(* CODESYS project distributedcontrol_1000.library
   Title: DistributedControl
   Version: 1.0.0.0
   Placeholder: DistributedControl
   Company: FactoryAutomation

Project tree, tasks and I/O mapping:
  libraries: Tc2_Standard, * (Beckhoff Automation GmbH); Tc2_System, * (Beckhoff Automation GmbH); Tc2_TcpIp, * (Beckhoff Automation GmbH); Tc3_Module, * (Beckhoff Automation GmbH)
  DUTs/
    data type E_TcpIpMode
    data type ST_ClientData
    data type ST_ServerData
  GVLs/
  POUs/
    program MAIN [ST]
    function block Payload [ST]
    function block Serializable [ST]: Deserialize, FB_exit, FB_init, Serialize
    function block TcpIp [ST]: FB_init, ReceiveSerializedObject, SendSerializedObject
  VISUs/
*)

// DUTs/E_TcpIpMode
TYPE E_TcpIpMode :
(
	TCP_IP_NO_MODE := 0,
	TCP_IP_SERVER,
	TCP_IP_CLIENT
);
END_TYPE

// DUTs/ST_ClientData
TYPE ST_ClientData :
STRUCT
	sSrvNetID   : T_AmsNetID := '';
    nMode       : DWORD := 0;
    sRemoteHost : T_IPv4Addr := '';
    nRemotePort : UDINT;
    tReconnect  : TIME := T#45S;
END_STRUCT
END_TYPE

// DUTs/ST_ServerData
TYPE ST_ServerData :
STRUCT
	hServer         : T_HSERVER; 
    sSrvNetID       : T_AmsNetID := ''; 
    sLocalHost      : STRING(15) := ''; 
    nLocalPort      : UDINT := 0;
	
    nMode           : DWORD := LISTEN_MODE_CLOSEALL (* OR CONNECT_MODE_ENABLEDBG*);
END_STRUCT
END_TYPE

// POUs/MAIN
PROGRAM MAIN
VAR

	fbPayload_1 : Payload(uiObjectSize := SIZEOF(Payload));
	fbPayload_2 : Payload(uiObjectSize := SIZEOF(Payload));
	
	bStart,
	bStart2,
	bStart3,
	bStart4,
	bStart5,
	bStart6 : BOOL;
	
	Size1,
	Size2,
	Size3,
	Size4 : UINT;
	pBuffer : POINTER TO BYTE;
	pServerBuffer : POINTER TO BYTE;
	pClientBuffer : POINTER TO BYTE;
	aMarshalBuffer : ARRAY[0..1999] OF BYTE;
	aServerMarshalBuffer : ARRAY[0..1999] OF BYTE;
	aClientMarshalBuffer : ARRAY[0..1999] OF BYTE;
	aServerBuffer : ARRAY[0..1999] OF BYTE;
	aClientBuffer : ARRAY[0..1999] OF BYTE;
	fbServer : TcpIp(TCP_IP_SERVER);
	fbClient : TcpIp(TCP_IP_CLIENT);
	serverStep : UINT;
	clientStep : UINT;
	udiServerTimeToSend : UDINT;
	udiServerTimeToReceive : UDINT;
	udiServerTimeToSendTmp : UDINT;
	udiServerTimeToReceiveTmp : UDINT;
END_VAR


fbPayload_1();
fbPayload_2();
fbPayload_1.timer.PT := T#45S;
fbPayload_1.timer.IN := TRUE;

fbServer.stServerData.nLocalPort := 200;
fbServer(bEnable := TRUE);

fbClient.stClientData.nRemotePort := 200;
fbClient(bEnable := TRUE);

IF 	bStart
	THEN
		
	pBuffer := fbPayload_2.Deserialize(fbPayload_1.Serialize());
	bStart := FALSE;
	
END_IF

IF	bStart2
	THEN
	
	MEMCPY(ADR(aMarshalBuffer),fbPayload_1.Serialize(),fbPayload_1.uiObjectSize);
	bStart2 := FALSE;
	
END_IF

IF	bStart3
	THEN
	
	fbPayload_2.Deserialize(ADR(aMarshalBuffer));
	bStart3 := FALSE;
	
END_IF

IF	bStart4
	THEN
	
	MEMCPY(ADR(aMarshalBuffer),fbPayload_2.Serialize(),fbPayload_2.uiObjectSize);
	bStart2 := FALSE;
	
END_IF
(*
IF	bStart5
	THEN
	
	CASE serverStep OF
	
		0 :
			MEMCPY(ADR(aServerMarshalBuffer),fbPayload_1.Serialize(),fbPayload_1.uiObjectSize);
			serverStep := 10;
			
		10:
		
			udiServerTimeToSendTmp := udiServerTimeToSendTmp + 1;
 			IF 	fbServer.SendSerializedObject(pSrc := ADR(aServerMarshalBuffer), cbLen := fbPayload_1.uiObjectSize)
				THEN
				
				udiServerTimeToSend := udiServerTimeToSendTmp;
				udiServerTimeToSendTmp := 0;
				serverStep := 20;
				
			END_IF
			
		20: 
		
			udiServerTimeToReceiveTmp := udiServerTimeToReceiveTmp + 1;
			IF 	fbServer.ReceiveSerializedObject(pDest := ADR(aServerBuffer),cbLen := fbPayload_1.uiObjectSize)
				THEN
				
				udiServerTimeToReceive := udiServerTimeToReceiveTmp;
				udiServerTimeToReceiveTmp := 0;
				
				fbPayload_1.Deserialize(ADR(aServerBuffer));
				serverStep := 0;
			END_IF
		
	END_CASE

	CASE clientStep OF
	
		0 :
 			IF 	fbClient.ReceiveSerializedObject(pDest := ADR(aClientBuffer),cbLen := fbPayload_2.uiObjectSize)
				THEN
				
				fbPayload_2.Deserialize(ADR(aClientBuffer));
				MEMCPY(ADR(aClientMarshalBuffer),fbPayload_2.Serialize(),fbPayload_2.uiObjectSize);
				
				clientStep := 10;
				
			END_IF
			
		10: 
			IF 	fbClient.SendSerializedObject(pSrc := ADR(aClientMarshalBuffer), cbLen := fbPayload_2.uiObjectSize)
				THEN
				
				clientStep := 0;
			END_IF
		
	END_CASE

END_IF
*)

END_PROGRAM

// POUs/Payload
FUNCTION_BLOCK Payload EXTENDS Serializable
VAR_INPUT
	timer : TON;
END_VAR
VAR_OUTPUT
END_VAR
VAR
	k : INT;	
END_VAR

timer();

END_FUNCTION_BLOCK

// POUs/Serializable
{attribute 'enable_dynamic_creation'}
FUNCTION_BLOCK Serializable

VAR_OUTPUT
	uiObjectSize : UINT;
	nWrittenBytes : UDINT;
END_VAR

VAR
	pSerializableObject : POINTER TO BYTE;
END_VAR

METHOD Deserialize : POINTER TO BYTE;
VAR_INPUT
	 pSerialObject : POINTER TO BYTE;
END_VAR
MEMCPY(THIS,pSerialObject,uiObjectSize);
Deserialize := pSerialObject;
END_METHOD

METHOD FB_exit : BOOL
VAR_INPUT
	bInCopyCode : BOOL; // if TRUE, the exit method is called for exiting an instance that is copied afterwards (online change).
END_VAR
IF pSerializableObject <> 0
THEN
	__DELETE(pSerializableObject);
END_IF
END_METHOD

METHOD FB_init : BOOL
VAR_INPUT
	bInitRetains : BOOL; // if TRUE, the retain variables are initialized (warm start / cold start)
	bInCopyCode : BOOL;  // if TRUE, the instance afterwards gets moved into the copy code (online change)
	uiObjectSize : UINT;
END_VAR
THIS^.uiObjectSize := uiObjectSize;
END_METHOD

METHOD Serialize : POINTER TO BYTE;
VAR_INPUT
END_VAR
IF pSerializableObject = 0
THEN

	Serialize := __NEW(BYTE,uiObjectSize);
	nWrittenBytes := MEMCPY(Serialize,THIS,uiObjectSize);
	pSerializableObject := Serialize;
	
ELSE
	Serialize := pSerializableObject;
END_IF
END_METHOD

END_FUNCTION_BLOCK

// POUs/TcpIp
FUNCTION_BLOCK TcpIp
VAR_INPUT
	
	bEnable : BOOL;
	stServerData : ST_ServerData;
	stClientData : ST_ClientData;
END_VAR
VAR_OUTPUT
END_VAR
VAR

	fbClientServerConnection : FB_ClientServerConnection;
	fbServerClientConnection : FB_ServerClientConnection;
	fbSocketSend : FB_SocketSend;
	fbSocketReceive : FB_SocketReceive;
	
	stepSendRoutine : UINT;
	stepReceiveRoutine : UINT;
	eMode : E_TcpIpMode;
	hSocket : T_HSOCKET;
END_VAR


fbSocketSend(
	sSrvNetId:= , 
	hSocket:= hSocket, 
	cbLen:= , 
	pSrc:= , 
	bExecute:= , 
	tTimeout:= , 
	bBusy=> , 
	bError=> , 
	nErrId=> );
	
fbSocketReceive(
	sSrvNetId:= , 
	hSocket:= hSocket, 
	cbLen:= , 
	pDest:= , 
	bExecute:= , 
	tTimeout:= , 
	bBusy=> , 
	bError=> , 
	nErrId=> , 
	nRecBytes=> );

CASE eMode OF

	TCP_IP_SERVER:
		F_CreateServerHnd(
			sSrvNetID := stServerData.sSrvNetID,
			bEnable := bEnable,
			sLocalHost := stServerData.sLocalHost,
			nLocalPort := stServerData.nLocalPort,
			nMode := stServerData.nMode,
			hServer := stServerData.hServer
		);
			
		fbServerClientConnection(
			hServer:= stServerData.hServer,
			eMode:= , 
			sRemoteHost:= , 
			nRemotePort:= , 
			bEnable:= bEnable, 
			tReconnect:= , 
			bBusy=> , 
			bError=> , 
			nErrID=> , 
			hSocket=> , 
			eState=> );
			
		hSocket := fbServerClientConnection.hSocket;	
		
	TCP_IP_CLIENT:
	
		fbClientServerConnection(
			sSrvNetID:= stClientData.sSrvNetID, 
			nMode:= stClientData.nMode, 
			sRemoteHost:= stClientData.sRemoteHost, 
			nRemotePort:= stClientData.nRemotePort, 
			bEnable:= bEnable, 
			tReconnect:= stClientData.tReconnect, 
			bBusy=> , 
			bError=> , 
			nErrId=> , 
			hSocket=> , 
			eState=> );
			
		hSocket := fbClientServerConnection.hSocket;		
		
END_CASE

METHOD FB_init : BOOL
VAR_INPUT
	bInitRetains : BOOL; // if TRUE, the retain variables are initialized (warm start / cold start)
	bInCopyCode : BOOL;  // if TRUE, the instance afterwards gets moved into the copy code (online change)
	eMode : E_TcpIpMode;
END_VAR
THIS^.eMode := eMode;
END_METHOD

METHOD ReceiveSerializedObject : BOOL
VAR_INPUT
	cbLen      : UDINT;
   	pDest      : POINTER TO BYTE;
END_VAR
IF	fbClientServerConnection.eState = eSOCKET_CONNECTED
	OR fbServerClientConnection.eState = eSOCKET_CONNECTED
THEN
	CASE stepReceiveRoutine OF
	
		0: 
			fbSocketReceive.pDest := pDest;
			fbSocketReceive.cbLen := cbLen;
			fbSocketReceive.bExecute := TRUE;
			stepReceiveRoutine := 10;
			
		10:
		
			IF 	NOT fbSocketReceive.bBusy
				AND NOT fbSocketReceive.bError
				AND fbSocketReceive.nRecBytes > 0
				THEN
				
				fbSocketReceive.bExecute := FALSE;
				ReceiveSerializedObject := TRUE;
				stepReceiveRoutine := 0;
				
			END_IF
			
	END_CASE
END_IF
END_METHOD

METHOD SendSerializedObject : BOOL
VAR_INPUT
	cbLen      : UDINT;
    pSrc       : POINTER TO BYTE;
END_VAR
IF 	fbClientServerConnection.eState = eSOCKET_CONNECTED
	OR fbServerClientConnection.eState = eSOCKET_CONNECTED
THEN
	CASE stepSendRoutine OF
	
		0: 
		
			fbSocketSend.pSrc := pSrc;
			fbSocketSend.cbLen := cbLen;
			fbSocketSend.bExecute := TRUE;
			stepSendRoutine := 10;
			
		10:
		
			IF 	NOT fbSocketSend.bBusy
				AND NOT fbSocketSend.bError
				
				THEN
				
				fbSocketSend.bExecute := FALSE;
				SendSerializedObject := TRUE;
				stepSendRoutine := 0;
				
			END_IF
			
	END_CASE
END_IF
END_METHOD

END_FUNCTION_BLOCK
